Staubli VAL3: readLogin.pgx

program readLogin(num handle_, string& msg_[], bool& result_[])
  local num nChar
  local num nCount
begin
  // read characters from socket until ":" is received
  msg_=""
  do
    nCount=sioGet(sSocket[handle_],nChar)
    if (nCount>-1) and (nChar>=32)
      msg_=msg_+chr(nChar)
    endIf
    result_=nCount>-1
  until (chr(nChar)==":") or !result_
  if !result_
    errorCode[handle_]=9
  endIf
  if bDebug
    putln("readLogin: "+msg_)
  endIf
end
